{attribute 'qualified_only'}
VAR_GLOBAL
	DeltaCoords : ARRAY[0..20] OF Coords;
	XYCoords	: ARRAY[0..20] OF Coords;
	I_bTest	AT %I*:BOOL;
	bGantryVac AT %Q*:BOOL;
	bGantryDown AT %Q*:BOOL;
	bGantryUp AT %Q*:BOOL;
END_VAR

(* stored: Version 1.1.0.1, ProductVersion 3.1.4024.11
   GVL GVL: Id {c0b59f4c-f1a2-4141-a240-1ec2cdbcdbf6} *)
